// TIA Portal V15.1 export
// export: Created 2024-06-21T08:40:49.954229Z, ExportSetting WithDefaults, DisplayName Totally Integrated Automation Portal, DisplayVersion V15.1 Update 5, DisplayName TIA Portal Openness, DisplayVersion V15.1 Update 5, DisplayName SINAMICS Startdrive Advanced, DisplayVersion V15.1, DisplayName G130, G150, S120, S150, SINAMICS MV, S210, DisplayVersion V15.1, DisplayName G110M, G120, G120C, G120D, G120P, DisplayVersion V15.1, DisplayName STEP 7 Professional, DisplayVersion V15.1 Update 5, DisplayName STEP 7 Safety, DisplayVersion V15.1, DisplayName WinCC Professional, DisplayVersion V15.1 Update 5, DisplayName SIMATIC Visualization Architect, DisplayVersion V15.1
DATA_BLOCK "_209220CWP14SH01AndonHCall"   // DB1832
{ S7_Optimized_Access := 'TRUE' }
VERSION : 0.1
// stored: AutoNumber false, DBAccessibleFromOPCUA true, InstanceOfName LGBAndonHCall, InstanceOfType FB
"LGBAndonHCall"
   // VAR_INPUT
   //    I_HCall { ExternalAccessible := 'False'; ExternalVisible := 'False'; ExternalWritable := 'False'} : Bool;
   //    I_PartPresent { ExternalAccessible := 'False'; ExternalVisible := 'False'; ExternalWritable := 'False'} : Bool;
   //    C_HCallNumber { ExternalAccessible := 'False'; ExternalVisible := 'False'; ExternalWritable := 'False'} : Int;
   //    C_WorkStationNumber { ExternalAccessible := 'False'; ExternalVisible := 'False'; ExternalWritable := 'False'} : Int;
   // END_VAR
   // VAR_OUTPUT
   //    O_AndonActiveSignal { ExternalAccessible := 'False'; ExternalVisible := 'False'; ExternalWritable := 'False'} : Bool;
   //    O_AndonCycleStpAfter { ExternalAccessible := 'False'; ExternalVisible := 'False'; ExternalWritable := 'False'} : Bool;
   // END_VAR
   // VAR_IN_OUT
   //    IO_AndonDataExchange : "AndonDataExchangeVCG";
   //    H_HMI : "H_HMI";
   //    H_GBAndonHCal : "H_GBAndonHCall";
   // END_VAR
   // VAR RETAIN
   //    AndonActiveSignal { ExternalAccessible := 'False'; ExternalVisible := 'False'; ExternalWritable := 'False'} : Bool;
   // END_VAR
   // VAR
   //    AndonHCallDW { ExternalAccessible := 'False'; ExternalVisible := 'False'; ExternalWritable := 'False'} : DWord;
   // END_VAR
   // VAR RETAIN
   //    AndonHCallActiveBits { ExternalAccessible := 'False'; ExternalVisible := 'False'; ExternalWritable := 'False'} : Array[0..31] of Bool;
   // END_VAR
   // VAR
   //    LToggle_AndonHCall { ExternalAccessible := 'False'; ExternalVisible := 'False'; ExternalWritable := 'False'} : "LToggle";
   //    AndonHCallActive { ExternalAccessible := 'False'; ExternalVisible := 'False'; ExternalWritable := 'False'} : DWord;
   //    CorrectedHCallNumber { ExternalAccessible := 'False'; ExternalVisible := 'False'; ExternalWritable := 'False'} : Int;
   // END_VAR
BEGIN
END_DATA_BLOCK
